// TIA Portal project "1_IL_DL-PN1_TIA" (V14)

(* hardware
DEVICE "S7-1200-Station_1"  S7-1200 Station
   slot 0: "Baugruppenträger_0"  S7-1200 Rack  Rack  V1.0
   slot 1: "PLC_1"  CPU 1212C AC/DC/Rly  6ES7 212-1BE40-0XB0  V4.2
DEVICE "GSD-Geraet_1"  GSD.Device.PN
   slot 0: "Baugruppenträger"  Rack  V1.0
   slot 0: "dl-pn1"  DL-PN1  DL-PN1  1.00
      slot 0: "DL-PN1"  DL-PN1  1.00
      slot 1: "Interface"  Interface
         slot 1: "Port 1"  Port 1
   slot 1: "DL-PN1_1"  DL-PN1
      slot 0: "DL-PN1 Device"  DL-PN1 Device
   slot 2: "IL-1***_1"  IL-1***
      slot 0: "IL-1***"  IL-1***
*)

// ===== PLC "PLC_1"  CPU 1212C AC/DC/Rly =====

VAR_GLOBAL   // PLC tag table "Standard-Variablentabelle"
   "Busy READ" AT %M1.1 : Bool;
   "Busy WRITE" AT %M0.2 : Bool;
   "Done WRITE" AT %M0.1 : Bool;
   "Error READ" AT %M1.2 : Bool;
   "Error WRITE" AT %M0.3 : Bool;
   "Ext IN-Reaktion 1 IL1000" AT %E18.0 : Bool;
   "Ext IN-Reaktion 1 IL1050" AT %E25.0 : Bool;
   "Ext IN-Reaktion 2 IL1000" AT %E18.1 : Bool;
   "Ext IN-Reaktion 2 IL1050" AT %E25.1 : Bool;
   "Ext IN-Reaktion 3 IL1000" AT %E18.2 : Bool;
   "Ext IN-Reaktion 3 IL1050" AT %E25.2 : Bool;
   "Ext IN-Reaktion 4 IL1000" AT %E18.3 : Bool;
   "Ext IN-Reaktion 4 IL1050" AT %E25.3 : Bool;
   "Ext IN Anf. 1 IL1000" AT %A1.0 : Bool;
   "Ext IN Anf. 1 IL1050" AT %A2.0 : Bool;
   "Ext IN Anf. 2 IL1000" AT %A1.1 : Bool;
   "Ext IN Anf. 2 IL1050" AT %A2.1 : Bool;
   "Ext IN Anf. 3 IL1000" AT %A1.2 : Bool;
   "Ext IN Anf. 3 IL1050" AT %A2.2 : Bool;
   "Ext IN Anf. 4 IL1000" AT %A1.3 : Bool;
   "Ext IN Anf. 4 IL1050" AT %A2.3 : Bool;
   "Fehlerstatus IL1000" AT %E17.7 : Bool;
   "Fehlerstatus IL1050" AT %E24.4 : Bool;
   "GO IL1000" AT %E16.2 : Bool;
   "GO IL1050" AT %E23.2 : Bool;
   "HIGH IL1000" AT %E16.0 : Bool;
   "HIGH IL1050" AT %E23.0 : Bool;
   "Len" AT %MW10 : Word;
   "LOW IL1000" AT %E16.1 : Bool;
   "LOW IL1050" AT %E23.1 : Bool;
   "Messwert IL1000" AT %ED19 : DInt;
   "Messwert IL1050" AT %ED26 : DInt;
   "Messwert u Bereich IL1000" AT %E17.2 : Bool;
   "Messwert ü Bereich IL1000" AT %E17.3 : Bool;
   "Messwert u Bereich IL1050" AT %E24.2 : Bool;
   "Messwert ü Bereich IL1050" AT %E24.3 : Bool;
   "Messwert ungültig IL1050" AT %E24.1 : Bool;
   "Messwert ungültig IL1000" AT %E17.1 : Bool;
   "REQUEST _RDREC" AT %E136.0 : Bool;
   "REQUEST _WRREC" AT %E136.1 : Bool;
   "Status READ" AT %MD6 : DWord;
   "Status WRITE" AT %MD2 : DWord;
   "Valid READ" AT %M1.0 : Bool;
   "Value_READ" AT %MD10 : DWord;
   "Value_WRITE" AT %MD14 : DWord;
END_VAR

ORGANIZATION_BLOCK "Main"   // OB1, FBD, ProgramCycle
TITLE = "Main Program Sweep (Cycle)"
{ S7_Optimized_Access := 'TRUE' }
VERSION : 0.1
   VAR_INPUT
      Initial_Call : Bool;   // Initial call of this OB
      Remanence : Bool;   // =True, if remanent data are available
   END_VAR
BEGIN

REGION Network 1: ReadRecord
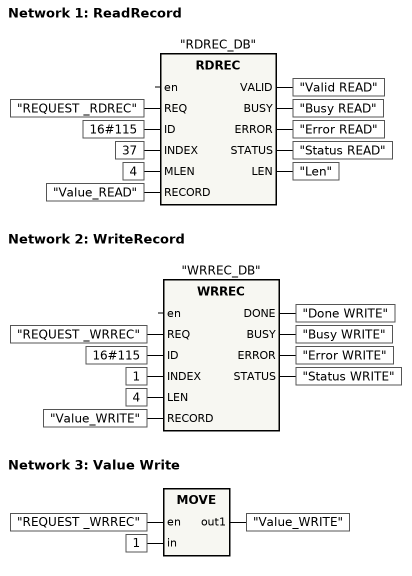
   "RDREC_DB"(REQ := "REQUEST _RDREC",   // RDREC
              ID := 16#115,
              INDEX := 37,
              MLEN := 4,
              RECORD := "Value_READ",
              VALID => "Valid READ",
              BUSY => "Busy READ",
              ERROR => "Error READ",
              STATUS => "Status READ",
              LEN => "Len");
END_REGION

REGION Network 2: WriteRecord
   "WRREC_DB"(REQ := "REQUEST _WRREC",   // WRREC
              ID := 16#115,
              INDEX := 1,
              LEN := 4,
              RECORD := "Value_WRITE",
              DONE => "Done WRITE",
              BUSY => "Busy WRITE",
              ERROR => "Error WRITE",
              STATUS => "Status WRITE");
END_REGION

REGION Network 3: Value Write
   IF "REQUEST _WRREC" THEN "Value_WRITE" := 1; END_IF;
END_REGION
END_ORGANIZATION_BLOCK